{attribute 'qualified_only'}
VAR_GLOBAL
END_VAR

(* stored: Version 1.1.0.1, ProductVersion 3.1.4022.7
   GVL SimAA: Id {62c4cdb6-e488-4cbf-8e50-e297ba05a31e} *)
